PROGRAM MAIN
VAR
	FB2_Counters : FB2_Counters;
	
END_VAR



FB2_Counters();
FC10_Alias();

END_PROGRAM

(* stored: Version 1.1.0.1, ProductVersion 3.1.4024.12
   POU MAIN: Id {45645433-dc31-41f0-b2c9-ed74135009fc}, SpecialFunc None *)
